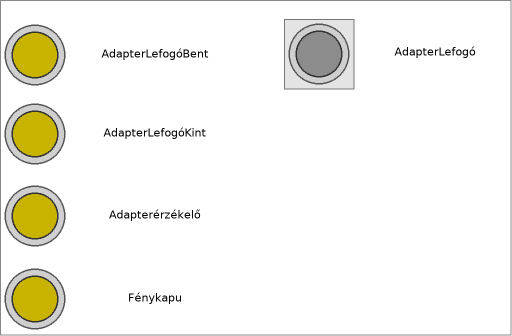
VISUALIZATION TempPistiBehelyezes  // 512x336
    Lamp1 (0,20 70x70), variable: GVL.bAdapterLefogoBent, style: Lamp-Lamp1-Yellow
    Label (80,39 150x30), "AdapterLefogóBent"
    Lamp1 (0,99 70x70), variable: GVL.bAdapterLefogoKint, style: Lamp-Lamp1-Yellow
    Label (80,118 150x30), "AdapterLefogóKint"
    Lamp1 (0,181 70x70), variable: GVL.bAdaptererzekelo, style: Lamp-Lamp1-Yellow
    Label (80,200 150x30), "Adapterérzékelő"
    Lamp1 (0,264 70x70), style: Lamp-Lamp1-Yellow
    Label (80,283 150x30), "Fénykapu"
    PushSwitch (284,19 70x70), variable: GVL.bAdapterLefogo, behaviour: TOGGLE, style: Switch-PushSwitch-Gray
    Label (360,37 150x30), "AdapterLefogó"
END_VISUALIZATION

(* stored: Version 1.1.0.1, ProductVersion 3.1.4024.11
   Visu TempPistiBehelyezes: Id {2f29ca11-daa5-4046-b1b4-112eda52cdc9} *)
